FUNCTION TryConvert_INT_TO_STRING : BOOL
VAR_INPUT
	in : INT;
	out : REFERENCE TO STRING;
END_VAR

out := INT_TO_STRING(in);
TryConvert_INT_TO_STRING := TRUE;

END_FUNCTION

(* stored: Version 1.1.0.1, ProductVersion 3.1.4024.12
   POU TryConvert_INT_TO_STRING: Id {b9461f56-6dde-4884-aee4-7e9b2c11611a}, SpecialFunc None *)
